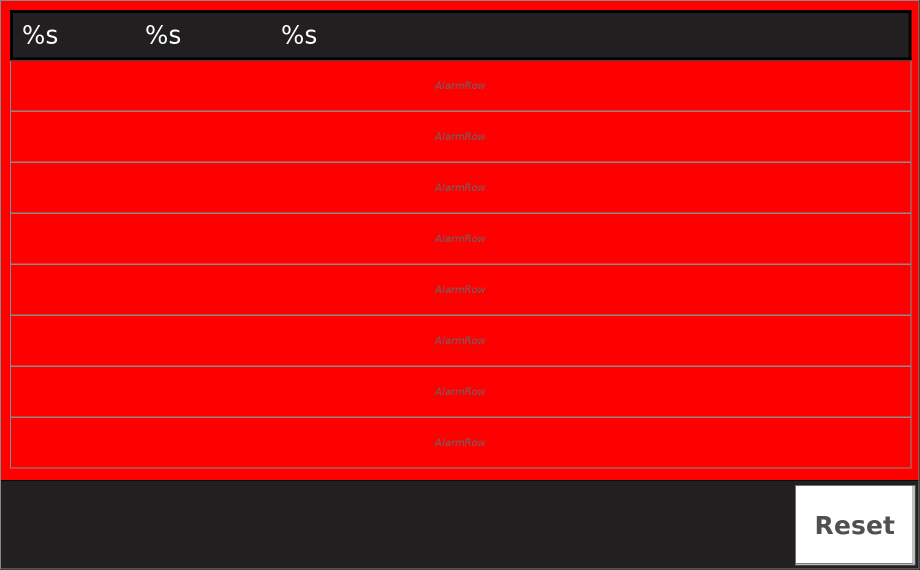
VISUALIZATION Alarm_Frame  // 920x570
VAR_IN_OUT
	xFaultResetPB : BOOL;
END_VAR

VAR_INPUT
	sAlarmTextList 	: STRING;
	sEventDataTextList : STRING;
	astActiveAlarmsList_1 : ST_AlarmEventData_TextList;
	astActiveAlarmsList_2 : ST_AlarmEventData_TextList;
	astActiveAlarmsList_3 : ST_AlarmEventData_TextList;
	astActiveAlarmsList_4 : ST_AlarmEventData_TextList;
	astActiveAlarmsList_5 : ST_AlarmEventData_TextList;
	astActiveAlarmsList_6 : ST_AlarmEventData_TextList;
	astActiveAlarmsList_7 : ST_AlarmEventData_TextList;
	astActiveAlarmsList_8 : ST_AlarmEventData_TextList;
END_VAR

VAR_OUTPUT
	
END_VAR
    Rectangle (0,0 920x570)
    Frame (10,60 901x51)
        shows AlarmRow(sAlarmTextList := sAlarmTextList, sEventDataTextList := sEventDataTextList, stAlarmLogEvent := astActiveAlarmsList_1)
    Frame (10,111 901x51)
        shows AlarmRow(sAlarmTextList := sAlarmTextList, sEventDataTextList := sEventDataTextList, stAlarmLogEvent := astActiveAlarmsList_2)
    Frame (10,213 901x51)
        shows AlarmRow(sAlarmTextList := sAlarmTextList, sEventDataTextList := sEventDataTextList, stAlarmLogEvent := astActiveAlarmsList_4)
    Frame (10,162 901x51)
        shows AlarmRow(sAlarmTextList := sAlarmTextList, sEventDataTextList := sEventDataTextList, stAlarmLogEvent := astActiveAlarmsList_3)
    Frame (10,264 901x51)
        shows AlarmRow(sAlarmTextList := sAlarmTextList, sEventDataTextList := sEventDataTextList, stAlarmLogEvent := astActiveAlarmsList_5)
    Frame (10,315 901x51)
        shows AlarmRow(sAlarmTextList := sAlarmTextList, sEventDataTextList := sEventDataTextList, stAlarmLogEvent := astActiveAlarmsList_6)
    Frame (10,366 901x51)
        shows AlarmRow(sAlarmTextList := sAlarmTextList, sEventDataTextList := sEventDataTextList, stAlarmLogEvent := astActiveAlarmsList_7)
    Frame (10,417 901x51)
        shows AlarmRow(sAlarmTextList := sAlarmTextList, sEventDataTextList := sEventDataTextList)
    Rectangle (10,10 901x50)
    Textfield (19,15 120x40), "%s", text list: sAlarmTextList, text index: 101
    Textfield (278,15 628x40), "%s", text list: sAlarmTextList, text index: 102
    Rectangle (0,480 920x90)
    Textfield (142,15 120x40), "%s", text list: sAlarmTextList, text index: 103
    Button (795,485 120x80), "Reset"
        tap xFaultResetPB
END_VISUALIZATION

(* stored: Version 1.1.0.1
   Visu Alarm_Frame: Id {6c1fe1b6-74db-4133-af22-16c8dc26d3da} *)
